RoboDK station: Conveying-and-Palletizing-with-Doosan-Robotics-H2017.rdk

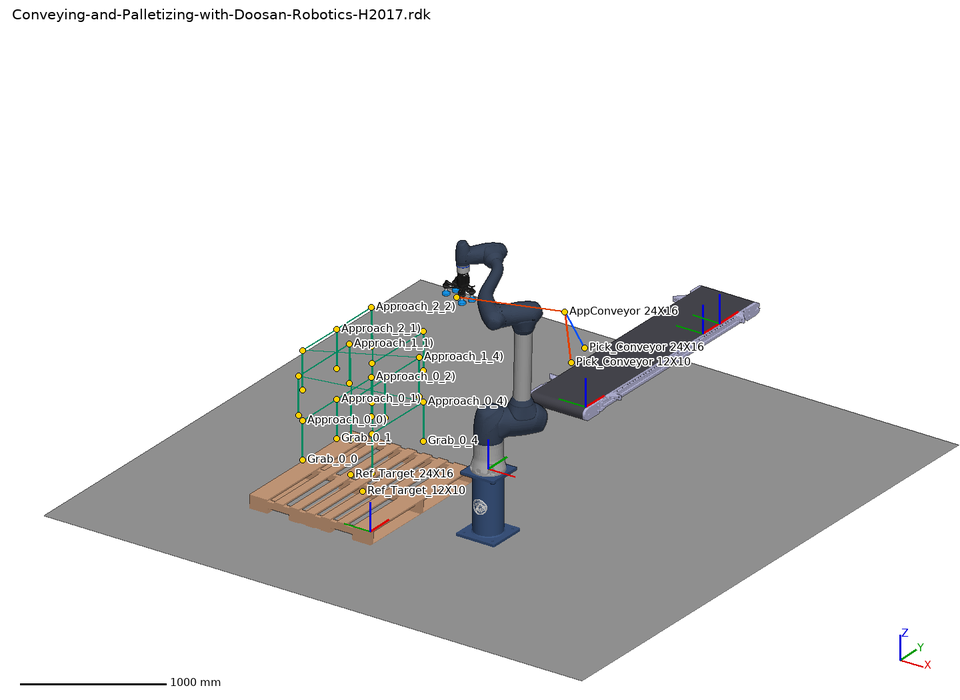
[picture v0: the station drawn from its stored meshes, robots at their saved joint values, targets as dots, program paths as lines]
Station Conveying and Palletizing with Doosan Robotics H2017 (saved by RoboDK 5.4.3). Poses are relative to the parent item; angles as X-Y-Z fixed-axis rotations.
Station parameters (name, value as stored): TAGS, ['Palletizing']
  - frame Doosan Robotics H2017 Base at (0, 0, 0) mm
    - object Pedestal H12in at (0, 0, -305) mm, rotated rx 0 ry 0 rz 90 deg, size 320 x 320 x 304.8 mm, geometry from Pedestal-H12in (2).sld
    - object Pedestal H24in at (0, 0, 0) mm, size 320 x 320 x 487.7 mm, geometry from Pedestal-H24in.sld
    - object Floor at (-410, 740, -496) mm, size 4500 x 4500 x 0 mm, geometry from Floor.sld
    - object Box 24X16 at (0, 0, 0) mm, size 398.1 x 610.2 x 267.5 mm, geometry from Box 24x16 closed.step
    - object Box 12X10 at (0, 0, 0) mm, size 252 x 305.4 x 216.7 mm, geometry from Box 12x10 closed.step
    - robot Doosan Robotics H2017: 6 axes, payload 20 kg, reach 1700 mm, repeatability 0.1 mm
        modified DH rows (alpha deg, a mm, theta deg, d mm): 0, 0, 180, 344.3; -90, 0, -90, -9.9; 0, 845, -90, 0; -90, 0, 0, 734; 90, 0, 0, 0; -90, 0, 180, 121
        joint limits [-360, -130, -160, -360, -360, -360] to [360, 130, 160, 360, 360, 360]; home [0, 0, -90, 0, -90, 0]; saved at [-38.939, 4.11, -84.5, 0, -99.61, 159.9]
      - tool RobotiQ EPick Four, TCP at (0, 30, 180) mm, size 239 x 147 x 184.9 mm
    - frame Pallet at (-556.43, -609.6, -390) mm, rotated rx 0 ry 0 rz 90 deg
      - object Pallet 40inx48in at (0, 0, 0) mm, size 1219.2 x 1016 x 114.3 mm, geometry from AR3.step
      - target Ref_Target_24X16 (Cartesian target) at (198.15, 304.16, 268.74) mm, rotated rx -180 ry 0 rz 90 deg; joints [27.742, -40.731, -104.765, 0, -34.504, 27.742] of Doosan Robotics H2017
      - target Ref_Target_12X10 (Cartesian target) at (125.28, 151.77, 216.13) mm, rotated rx -180 ry 0 rz 90 deg; joints [36.637, -40.651, -113.092, 0, -26.257, 36.637] of Doosan Robotics H2017
      - folder Palletizing Settings Data
        - folder Layer 0
          - target Approach_0_0) (Cartesian target) at (198.91, 708.58, 567.5) mm, rotated rx -180 ry 0 rz 89.86 deg; joints [18.413, -53.81, -64.204, 0, -61.986, 18.55] of Doosan Robotics H2017
          - target Grab_0_0 (Cartesian target) at (198.91, 708.58, 267.5) mm, rotated rx -180 ry 0 rz 89.86 deg; joints [18.413, -66.621, -64.333, 0, -49.046, 18.55] of Doosan Robotics H2017
          - target Approach_0_1) (Cartesian target) at (608.41, 708.58, 567.5) mm, rotated rx -180 ry 0 rz 89.86 deg; joints [0.502, -49.71, -72.591, 0, -57.699, 0.639] of Doosan Robotics H2017
          - target Grab_0_1 (Cartesian target) at (608.41, 708.58, 267.5) mm, rotated rx -180 ry 0 rz 89.86 deg; joints [0.502, -63.181, -72.713, 0, -44.107, 0.639] of Doosan Robotics H2017
          - target Approach_0_2) (Cartesian target) at (1024.41, 708.58, 567.5) mm, rotated rx -180 ry 0 rz 89.86 deg; joints [-17.729, -53.894, -64.03, 0, -62.076, -17.592] of Doosan Robotics H2017
          - target Grab_0_2 (Cartesian target) at (1024.41, 708.58, 267.5) mm, rotated rx -180 ry 0 rz 89.86 deg; joints [-17.729, -66.694, -64.159, 0, -49.147, -17.592] of Doosan Robotics H2017
          - target Approach_0_3) (Cartesian target) at (305.58, 200.16, 567.5) mm, rotated rx -180 ry 0 rz -0.09 deg; joints [22.588, -27.313, -117.057, 0, -35.63, 112.679] of Doosan Robotics H2017
          - target Grab_0_3 (Cartesian target) at (305.58, 200.16, 267.5) mm, rotated rx -180 ry 0 rz -0.09 deg; joints [22.588, -48.113, -117.188, 180, 14.699, -67.321] of Doosan Robotics H2017
          - target Approach_0_4) (Cartesian target) at (916.58, 200.16, 567.5) mm, rotated rx -180 ry 0 rz -0.09 deg; joints [-21.39, -27.362, -116.963, 0, -35.675, 68.702] of Doosan Robotics H2017
          - target Grab_0_4 (Cartesian target) at (916.58, 200.16, 267.5) mm, rotated rx -180 ry 0 rz -0.09 deg; joints [-21.39, -48.134, -117.094, 0, -14.772, 68.702] of Doosan Robotics H2017
        - folder Layer 1
          - target Approach_1_0) (Cartesian target) at (305.58, 817.66, 835) mm, rotated rx -180 ry 0 rz -0.09 deg; joints [12.879, -53.351, -43.117, 0, -83.532, 102.97] of Doosan Robotics H2017
          - target Grab_1_0 (Cartesian target) at (305.58, 817.66, 535) mm, rotated rx -180 ry 0 rz -0.09 deg; joints [12.879, -60.458, -53.234, 0, -66.308, 102.97] of Doosan Robotics H2017
          - target Approach_1_1) (Cartesian target) at (916.58, 817.66, 835) mm, rotated rx -180 ry 0 rz -0.09 deg; joints [-12.191, -53.415, -42.995, 0, -83.591, 77.901] of Doosan Robotics H2017
          - target Grab_1_1 (Cartesian target) at (916.58, 817.66, 535) mm, rotated rx -180 ry 0 rz -0.09 deg; joints [-12.191, -60.508, -53.13, 0, -66.362, 77.901] of Doosan Robotics H2017
          - target Approach_1_2) (Cartesian target) at (198.91, 305.58, 835) mm, rotated rx -180 ry 0 rz 89.86 deg; joints [26.069, -21.976, -97.566, 0, -60.458, 26.206] of Doosan Robotics H2017
          - target Grab_1_2 (Cartesian target) at (198.91, 305.58, 535) mm, rotated rx -180 ry 0 rz 89.86 deg; joints [26.069, -35.368, -105.253, 0, -39.379, 26.206] of Doosan Robotics H2017
          - target Approach_1_3) (Cartesian target) at (608.41, 305.58, 835) mm, rotated rx -180 ry 0 rz 89.86 deg; joints [0.737, -16.452, -105.524, 0, -58.024, 0.874] of Doosan Robotics H2017
          - target Grab_1_3 (Cartesian target) at (608.41, 305.58, 535) mm, rotated rx -180 ry 0 rz 89.86 deg; joints [0.737, -31.326, -113.519, 0, -35.155, 0.874] of Doosan Robotics H2017
          - target Approach_1_4) (Cartesian target) at (1017.91, 305.58, 835) mm, rotated rx -180 ry 0 rz 89.86 deg; joints [-24.751, -21.915, -97.657, 0, -60.428, -24.614] of Doosan Robotics H2017
          - target Grab_1_4 (Cartesian target) at (1017.91, 305.58, 535) mm, rotated rx -180 ry 0 rz 89.86 deg; joints [-24.751, -35.322, -105.347, 0, -39.331, -24.614] of Doosan Robotics H2017
        - folder Layer 2
          - target Approach_2_0) (Cartesian target) at (198.91, 708.58, 1102.5) mm, rotated rx -180 ry 0 rz 89.86 deg; joints [18.413, -45.466, -36.973, 0, -97.561, 18.55] of Doosan Robotics H2017
          - target Grab_2_0 (Cartesian target) at (198.91, 708.58, 802.5) mm, rotated rx -180 ry 0 rz 89.86 deg; joints [18.413, -47.172, -57.445, 0, -75.383, 18.55] of Doosan Robotics H2017
          - target Approach_2_1) (Cartesian target) at (608.41, 708.58, 1102.5) mm, rotated rx -180 ry 0 rz 89.86 deg; joints [0.502, -38.992, -48.475, 0, -92.533, 0.639] of Doosan Robotics H2017
          - target Grab_2_1 (Cartesian target) at (608.41, 708.58, 802.5) mm, rotated rx -180 ry 0 rz 89.86 deg; joints [0.502, -42.382, -66.288, 0, -71.33, 0.639] of Doosan Robotics H2017
          - target Approach_2_2) (Cartesian target) at (1024.41, 708.58, 1102.5) mm, rotated rx -180 ry 0 rz 89.86 deg; joints [-17.729, -45.609, -36.712, 0, -97.679, -17.592] of Doosan Robotics H2017
          - target Grab_2_2 (Cartesian target) at (1024.41, 708.58, 802.5) mm, rotated rx -180 ry 0 rz 89.86 deg; joints [-17.729, -47.271, -57.259, 0, -75.47, -17.592] of Doosan Robotics H2017
          - target Approach_2_3) (Cartesian target) at (305.58, 200.16, 1102.5) mm, rotated rx -180 ry 0 rz -0.09 deg; joints [22.588, -6.582, -95.228, 0, -78.19, 112.679] of Doosan Robotics H2017
          - target Grab_2_3 (Cartesian target) at (305.58, 200.16, 802.5) mm, rotated rx -180 ry 0 rz -0.09 deg; joints [22.588, -14.977, -110.605, 0, -54.418, 112.679] of Doosan Robotics H2017
          - target Approach_2_4) (Cartesian target) at (916.58, 200.16, 1102.5) mm, rotated rx -180 ry 0 rz -0.09 deg; joints [-21.39, -6.656, -95.144, 0, -78.2, 68.702] of Doosan Robotics H2017
          - target Grab_2_4 (Cartesian target) at (916.58, 200.16, 802.5) mm, rotated rx -180 ry 0 rz -0.09 deg; joints [-21.39, -15.042, -110.516, 0, -54.441, 68.702] of Doosan Robotics H2017
    - frame Conveyor Belt Base at (430, 550, 370) mm, rotated rx 0 ry 0 rz 90 deg
      - robot Conveyor Belt: 1 axes
          modified DH rows (alpha deg, a mm, theta deg, d mm): 0, 0, 0, 0 linear
          base shift (0, 0, 0) mm, rotated rx 0 ry 90 rz 0 deg
          joint limits [-500000] to [500000]; home [0]; saved at [0]
        - frame Conveyor Box at (0, 0, 0) mm
      - target AppConveyor 24X16 (Cartesian target) at (69.16, 222.69, 638.74) mm, rotated rx 180 ry 0 rz 179.98 deg; joints [-110.116, 4.118, -84.501, 0, -99.617, 159.905, 0] of Doosan Robotics H2017
      - target Pick_Conveyor 24X16 (Cartesian target) at (304.16, 222.6, 268.74) mm, rotated rx 180 ry 0 rz 179.98 deg; joints [-104.892, -12.914, -95.198, 0, -71.888, 165.128, 0] of Doosan Robotics H2017
      - target AppConveyor 12X10 (Cartesian target) at (69.16, 222.69, 638.74) mm, rotated rx 180 ry 0 rz 179.98 deg; joints [-110.116, 4.118, -84.501, 0, -99.617, 159.905] of Doosan Robotics H2017
      - target Pick_Conveyor 12X10 (Cartesian target) at (151.76, 228.42, 216.13) mm, rotated rx 180 ry 0 rz 179.98 deg; joints [-107.495, -4.666, -109.405, 0, -65.929, 162.525] of Doosan Robotics H2017
      - target Trans_Conveyor (Cartesian target) at (-168.56, 960.11, 638.66) mm, rotated rx 180 ry 0 rz -107.24 deg; joints [-37.34, 4.11, -84.5, 0, -99.61, 159.9] of Doosan Robotics H2017
      - frame New_Box 24X16 at (1400, 0, 0) mm
        - object BoxRef_24X16 at (0, 420, 0) mm, rotated rx 0 ry 0 rz -90 deg, size 398.1 x 610.2 x 267.5 mm, geometry from Box 24x16 closed.step
      - frame New_Box 12X10 at (1600, 0, 0) mm
        - object BoxRef_12X10 at (0, 350, 0) mm, rotated rx 0 ry 0 rz -90 deg, size 252 x 305.4 x 216.7 mm, geometry from Box 12x10 closed.step
    - object Box 24X16 at (0, 0, 0) mm, size 398.1 x 610.2 x 267.5 mm, geometry from Box 24x16 closed.step
  - program Pick_Box_24X16 (10 instructions, listed below)
  - program Pick_Box_12X10 (10 instructions, listed below)
  - item type 20 Palletizing Settings: svg | Palletizing Plugin | Pallet | Conveyor Belt | Box 24X16 | Box 24X16 | Box 24X16 | Box 24X16 | Init_24X16 | Pick_Box_24X16 | Drop_Box | onLayer(%1) | onFinish
  - program Init_24X16 (8 instructions, listed below)
  - program Drop_Box (1 instructions, listed below)
  - folder Python
    - Python program Clear_Conveyor (listed below)
    - Python program Clear_Pallet (listed below)
    - Python program Clear_Tool (listed below)
    - Python program Conv_Init_Position (listed below)
    - Python program Conv_Move_24X16 (listed below)
    - Python program Conv_Move_12X10 (listed below)
    - Python program New_Box_12X10 (listed below)
    - Python program New_Box_24X16 (listed below)
  - program Main (108 instructions, listed below)
  - program Reset (4 instructions, listed below)
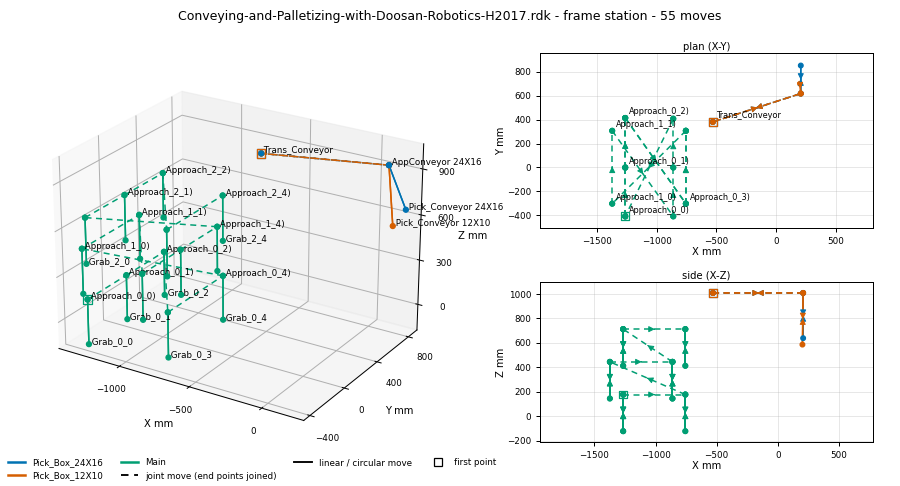
[picture p0: tool path of Conveying-and-Palletizing-with-Doosan-Robotics-H2017.rdk in frame station, 55 of 55 moves have a stored position in this frame; points joined in program order, loops and branches not executed]

--- program Pick_Box_24X16 (robot Doosan Robotics H2017) ---
  Set Ref.: Conveyor Belt Base
  Set Tool: RobotiQ EPick Four
  Call New_Box_24X16
  MoveJ (Trans_Conveyor)
  MoveJ (AppConveyor 24X16)
  MoveL (Pick_Conveyor 24X16)
  Attach to RobotiQ EPick Four
  MoveL (AppConveyor 24X16)
  Run Conv_Move_24X16
  MoveJ (Trans_Conveyor)

--- program Pick_Box_12X10 (robot Doosan Robotics H2017) ---
  Set Ref.: Conveyor Belt Base
  Set Tool: RobotiQ EPick Four
  Call New_Box_12X10
  MoveJ (Trans_Conveyor)
  MoveJ (AppConveyor 12X10)
  MoveL (Pick_Conveyor 12X10)
  Attach to RobotiQ EPick Four
  MoveL (AppConveyor 12X10)
  Run Conv_Move_24X16
  MoveJ (Trans_Conveyor)

--- program Init_24X16 (robot Doosan Robotics H2017) ---
  Call Conv_Init_Position
  Call Clear_Conveyor
  Call Clear_Pallet
  Call Clear_Tool
  Call New_Box_24X16
  Call Conv_Move_24X16
  Call New_Box_24X16
  Call Conv_Move_24X16

--- program Drop_Box (robot Doosan Robotics H2017) ---
  Detach from RobotiQ EPick Four

--- Python program Clear_Conveyor ---
# Type help("robolink") or help("robodk") for more information
# Press F5 to run the script
# Documentation: https://robodk.com/doc/en/RoboDK-API.html
# Reference:     https://robodk.com/doc/en/PythonAPI/index.html
# Note: It is not required to keep a copy of this file, your python script is saved with the station
from robodk import robolink
RDK = robolink.Robolink()

#----- CONSTANT -----
CONV_FRAME_NAME = 'Conveyor Box'

#----- PROGRAM -----
frame = RDK.Item(CONV_FRAME_NAME,robolink.ITEM_TYPE_FRAME)

if frame.Valid():
    for item in frame.Childs():
        if item.Type() == robolink.ITEM_TYPE_OBJECT:
            item.Delete()

--- Python program Clear_Pallet ---
# Type help("robolink") or help("robodk") for more information
# Press F5 to run the script
# Documentation: https://robodk.com/doc/en/RoboDK-API.html
# Reference:     https://robodk.com/doc/en/PythonAPI/index.html
# Note: It is not required to keep a copy of this file, your python script is saved with the station
from robodk import robolink
RDK = robolink.Robolink()

#----- CONSTANT -----
FRAME_NAME = 'Pallet'

#----- PROGRAM -----
frame = RDK.Item(FRAME_NAME,robolink.ITEM_TYPE_FRAME)

if frame.Valid():
    for item in frame.Childs():
        if item.Type() == robolink.ITEM_TYPE_OBJECT:
            if not item.Name().lower().startswith('pallet'):
                item.Delete()

--- Python program Clear_Tool ---
# Type help("robolink") or help("robodk") for more information
# Press F5 to run the script
# Documentation: https://robodk.com/doc/en/RoboDK-API.html
# Reference:     https://robodk.com/doc/en/PythonAPI/index.html
# Note: It is not required to keep a copy of this file, your python script is saved with the station

from robodk import robolink
RDK = robolink.Robolink()

#----- CONSTANT -----
TOOL_NAME = 'RobotiQ EPick Four'

#----- PROGRAM -----
tool = RDK.Item(TOOL_NAME, robolink.ITEM_TYPE_FRAME)

if tool.Valid():
    for item in tool.Childs():
        if item.Type() == robolink.ITEM_TYPE_OBJECT:
            item.Delete()

--- Python program Conv_Init_Position ---
# Type help("robolink") or help("robodk") for more information
# Press F5 to run the script
# Documentation: https://robodk.com/doc/en/RoboDK-API.html
# Reference:     https://robodk.com/doc/en/PythonAPI/index.html
# Note: It is not required to keep a copy of this file, your python script is saved with the station
from robodk import robolink
RDK = robolink.Robolink()

MECHANISM_NAME = 'Conveyor Belt'

mechanism = RDK.Item(MECHANISM_NAME,itemtype=robolink.ITEM_TYPE_ROBOT)

if mechanism.Valid():
    mechanism.setJoints([0])

--- Python program Conv_Move_24X16 ---
# Type help("robolink") or help("robodk") for more information
# Press F5 to run the script
# Documentation: https://robodk.com/doc/en/RoboDK-API.html
# Reference:     https://robodk.com/doc/en/PythonAPI/index.html
# Note: It is not required to keep a copy of this file, your python script is saved with the station
from robodk import robolink
RDK = robolink.Robolink()

#------ CONSTANT ------
MECHANISM_NAME = 'Conveyor Belt'
PART_TRAVEL_MM = -700

mechanism = RDK.Item(MECHANISM_NAME,itemtype=robolink.ITEM_TYPE_ROBOT)

if mechanism.Valid():
    mechanism.MoveJ(mechanism.Joints() + PART_TRAVEL_MM)

--- Python program Conv_Move_12X10 ---
# Type help("robolink") or help("robodk") for more information
# Press F5 to run the script
# Documentation: https://robodk.com/doc/en/RoboDK-API.html
# Reference:     https://robodk.com/doc/en/PythonAPI/index.html
# Note: It is not required to keep a copy of this file, your python script is saved with the station
from robodk import robolink
RDK = robolink.Robolink()

#------ CONSTANT ------
MECHANISM_NAME = 'Conveyor Belt'
PART_TRAVEL_MM = -400

mechanism = RDK.Item(MECHANISM_NAME,itemtype=robolink.ITEM_TYPE_ROBOT)

if mechanism.Valid():
    mechanism.MoveJ(mechanism.Joints() + PART_TRAVEL_MM)

--- Python program New_Box_12X10 ---
# Type help("robolink") or help("robodk") for more information
# Press F5 to run the script
# Documentation: https://robodk.com/doc/en/RoboDK-API.html
# Reference:     https://robodk.com/doc/en/PythonAPI/index.html
# Note: It is not required to keep a copy of this file, your python script is saved with the station
from robodk import robolink
RDK = robolink.Robolink()

#----- Constante -----
NEW_REF_OBJECT_NAME = 'BoxRef_12X10'
NEW_OBJECT_NAME = 'Box_12X10'
REFERENCE_FRAME = 'Conveyor Box'
REFERENCE_FRAME_REF = 'New_Box 12X10'


#------- Program ------
frame = RDK.Item(REFERENCE_FRAME, robolink.ITEM_TYPE_FRAME)
frame_ref = RDK.Item(REFERENCE_FRAME_REF, robolink.ITEM_TYPE_FRAME)
ref_obj = RDK.Item(NEW_REF_OBJECT_NAME, robolink.ITEM_TYPE_OBJECT)

if frame.Valid() and  ref_obj.Valid():
    ref_obj.Copy()
    new_obj = RDK.Paste()
    new_obj.setVisible(False)
    new_obj.setName(NEW_OBJECT_NAME)
    new_obj.setParent(frame_ref)
    new_obj.setParentStatic(frame)
    new_obj.setVisible(True)

--- Python program New_Box_24X16 ---
# Type help("robolink") or help("robodk") for more information
# Press F5 to run the script
# Documentation: https://robodk.com/doc/en/RoboDK-API.html
# Reference:     https://robodk.com/doc/en/PythonAPI/index.html
# Note: It is not required to keep a copy of this file, your python script is saved with the station
from robodk import robolink
RDK = robolink.Robolink()

#----- Constante -----
NEW_REF_OBJECT_NAME = 'BoxRef_24X16'
NEW_OBJECT_NAME = 'Box_24X16'
REFERENCE_FRAME = 'Conveyor Box'
REFERENCE_FRAME_REF = 'New_Box 24X16'


#------- Program ------
frame = RDK.Item(REFERENCE_FRAME, robolink.ITEM_TYPE_FRAME)
frame_ref = RDK.Item(REFERENCE_FRAME_REF, robolink.ITEM_TYPE_FRAME)
ref_obj = RDK.Item(NEW_REF_OBJECT_NAME, robolink.ITEM_TYPE_OBJECT)

if frame.Valid() and  ref_obj.Valid():
    ref_obj.Copy()
    new_obj = RDK.Paste()
    new_obj.setVisible(False)
    new_obj.setName(NEW_OBJECT_NAME)
    new_obj.setParent(frame_ref)
    new_obj.setParentStatic(frame)
    new_obj.setVisible(True)

--- program Main (robot Doosan Robotics H2017) ---
  Set Ref.: Pallet
  Call Init_24X16
  Set Ref.: Pallet
  Call Pick_Box_24X16
  Set Ref.: Pallet
  MoveJ (Approach_0_0))
  MoveL (Grab_0_0)
  Call Drop_Box
  Set Ref.: Pallet
  MoveL (Approach_0_0))
  Call Pick_Box_24X16
  Set Ref.: Pallet
  MoveJ (Approach_0_1))
  MoveL (Grab_0_1)
  Call Drop_Box
  Set Ref.: Pallet
  MoveL (Approach_0_1))
  Call Pick_Box_24X16
  Set Ref.: Pallet
  MoveJ (Approach_0_2))
  MoveL (Grab_0_2)
  Call Drop_Box
  Set Ref.: Pallet
  MoveL (Approach_0_2))
  Call Pick_Box_24X16
  Set Ref.: Pallet
  MoveJ (Approach_0_3))
  MoveL (Grab_0_3)
  Call Drop_Box
  Set Ref.: Pallet
  MoveL (Approach_0_3))
  Call Pick_Box_24X16
  Set Ref.: Pallet
  MoveJ (Approach_0_4))
  MoveL (Grab_0_4)
  Call Drop_Box
  Set Ref.: Pallet
  MoveL (Approach_0_4))
  Call Pick_Box_24X16
  Set Ref.: Pallet
  MoveJ (Approach_1_0))
  MoveL (Grab_1_0)
  Call Drop_Box
  Set Ref.: Pallet
  MoveL (Approach_1_0))
  Call Pick_Box_24X16
  Set Ref.: Pallet
  MoveJ (Approach_1_1))
  MoveL (Grab_1_1)
  Call Drop_Box
  Set Ref.: Pallet
  MoveL (Approach_1_1))
  Call Pick_Box_24X16
  Set Ref.: Pallet
  MoveJ (Approach_1_2))
  MoveL (Grab_1_2)
  Call Drop_Box
  Set Ref.: Pallet
  MoveL (Approach_1_2))
  Call Pick_Box_24X16
  Set Ref.: Pallet
  MoveJ (Approach_1_3))
  MoveL (Grab_1_3)
  Call Drop_Box
  Set Ref.: Pallet
  MoveL (Approach_1_3))
  Call Pick_Box_24X16
  Set Ref.: Pallet
  MoveJ (Approach_1_4))
  MoveL (Grab_1_4)
  Call Drop_Box
  Set Ref.: Pallet
  MoveL (Approach_1_4))
  Call Pick_Box_24X16
  Set Ref.: Pallet
  MoveJ (Approach_2_0))
  MoveL (Grab_2_0)
  Call Drop_Box
  Set Ref.: Pallet
  MoveL (Approach_2_0))
  Call Pick_Box_24X16
  Set Ref.: Pallet
  MoveJ (Approach_2_1))
  MoveL (Grab_2_1)
  Call Drop_Box
  Set Ref.: Pallet
  MoveL (Approach_2_1))
  Call Pick_Box_24X16
  Set Ref.: Pallet
  MoveJ (Approach_2_2))
  MoveL (Grab_2_2)
  Call Drop_Box
  Set Ref.: Pallet
  MoveL (Approach_2_2))
  Call Pick_Box_24X16
  Set Ref.: Pallet
  MoveJ (Approach_2_3))
  MoveL (Grab_2_3)
  Call Drop_Box
  Set Ref.: Pallet
  MoveL (Approach_2_3))
  Call Pick_Box_24X16
  Set Ref.: Pallet
  MoveJ (Approach_2_4))
  MoveL (Grab_2_4)
  Call Drop_Box
  Set Ref.: Pallet
  MoveL (Approach_2_4))

--- program Reset (robot Doosan Robotics H2017) ---
  Call Clear_Conveyor
  Call Clear_Pallet
  Call Clear_Tool
  Call Conv_Init_Position
